// TwinCAT 3 PLC project Este_es_el_PLC
// ProgramVersion: 3.1.4024.0
// libraries:
//   Tc2_EtherCAT, * (Beckhoff Automation GmbH)
//   Tc2_ModbusSrv, * (Beckhoff Automation GmbH)
//   Tc2_Standard, * (Beckhoff Automation GmbH)
//   Tc2_System, * (Beckhoff Automation GmbH)
//   Tc2_Utilities, * (Beckhoff Automation GmbH)
//   Tc3_Module, * (Beckhoff Automation GmbH)
// project tree:
//   DUTs/ E_EventType.TcDUT, St_Event.TcDUT, ST_MachineStation.TcDUT (not stored)
//   GVLs/ GVL.TcGVL, Tags.TcGVL
//   / PlcTask.TcTTO
//   POUs/ conveyor1.TcPOU, MAIN.TcPOU
// real-time tasks:
//   TASK PlcTask: cycle T#10ms, priority 20, ADS port 350
//   TASK Device 1 (OPC UA Virtual)_Task_58: cycle T#40ms, priority 58, ADS port 351

CONFIGURATION Este_es_el_PLC
    RESOURCE PLC ON TwinCAT3
        TASK PlcTask(INTERVAL := T#10ms, PRIORITY := 20);
        PROGRAM MAIN WITH PlcTask : MAIN;
    END_RESOURCE
END_CONFIGURATION

// ---- DUTs/E_EventType.TcDUT
{attribute 'qualified_only'}
{attribute 'strict'}
TYPE E_EventType :
(
	alarm := 0,
	Message := 1
);
END_TYPE

// ---- DUTs/St_Event.TcDUT
TYPE St_Event :
STRUCT
	eEventType : E_EventType;
	eVentSeverity : TcEventSeverity;
	nEventIdentity : UDINT;
	SEventText : STRING(255);
	dtTimeStamp : DATE_AND_TIME;
END_STRUCT
END_TYPE

// ---- GVLs/GVL.TcGVL
{attribute 'qualified_only'}
VAR_GLOBAL
	mb_Input_Coils : ARRAY [0..255] OF BOOL;
	mb_Output_Coils : ARRAY [0..255] OF BOOL;
	mb_Input_Registers : ARRAY [0..255] OF WORD;
	mb_Output_Registers : ARRAY [0..255] OF WORD;
END_VAR

// ---- GVLs/Tags.TcGVL
{attribute 'qualified_only'}
VAR_GLOBAL
	bAutoMan : SR;
END_VAR

// ---- POUs/MAIN.TcPOU
PROGRAM MAIN
VAR
	bButtonStart,
	bButtonReset,
	bButtonStop: BOOL;
	bStatus : BOOL;
	bButtonLightStart,
	bButtonLightStop,
	bExtra, botroextra,bTercer,bCuarto : BOOL;
END_VAR

bButtonStart := GVL.mb_Output_Coils[0];
bButtonStop := GVL.mb_Output_Coils[1];
bButtonReset := GVL.mb_Output_Coils[29];
GVL.mb_Input_Coils[0] := bButtonLightStart;
GVL.mb_Input_Coils[1] := bButtonLightStop;
conveyor1();

Tags.bAutoMan(SET1 := bButtonStart, RESET := NOT bButtonStop);
bStatus := Tags.bAutoMan.Q1;
bButtonLightStart := bStatus;
bButtonLightStop := not bStatus;

END_PROGRAM

// ---- POUs/conveyor1.TcPOU
PROGRAM conveyor1
VAR
	bStatus: BOOL;
	bSensor2: BOOL;
	bSensor1: BOOL;
	bAlimentador1: BOOL;
	intCaseConveyor : INT;
	bButtonReset: BOOL;
	timer1, timer2, timer3,timer4 : TON;
	bConvFowar1: BOOL;
	bMachineCenterOpen: BOOL;
	bMachineCenterBusy: BOOL;
	bStartMachineCenter: BOOL;
	wMachineProgress: WORD;
END_VAR

bStatus := tags.bAutoMan.Q1;
bSensor1 := GVL.mb_Output_Coils[10];
bSensor2 := GVL.mb_Output_Coils[11];
bButtonReset := gvl.mb_Output_Coils[2];
bMachineCenterOpen := gvl.mb_Output_Coils[12];
bMachineCenterBusy := gvl.mb_Output_Coils[13];
wMachineProgress := gvl.mb_Output_Registers[0];


GVL.mb_Input_Coils[10] := bAlimentador1;
GVL.mb_Input_Coils[11] := bConvFowar1;
GVL.mb_Input_Coils[12] := bStartMachineCenter;

timer1(PT:= T#1S);
timer2(PT:= T#1S);
timer3(PT:= T#1S);


IF NOT bStatus THEN
	intCaseConveyor := 0;
END_IF

IF intCaseConveyor = 40 THEN
	timer2(IN := TRUE);
ELSE
	timer2(IN := FALSE);
END_IF

IF intCaseConveyor = 50 THEN
	timer3(IN := TRUE);
ELSE
	timer3(IN := FALSE);
END_IF

CASE intCaseConveyor OF
	00: timer1(IN:= FALSE);
		timer4(IN:= FALSE);
		bConvFowar1 := FALSE;
		bStartMachineCenter := False;
		IF bStatus THEN
			IF bSensor1 THEN
				intCaseConveyor := 10;
			ELSE
				intCaseConveyor := 20;
			END_IF
		END_IF
	10: IF bSensor1 THEN
			bAlimentador1 := TRUE;
		ELSE
			bAlimentador1 := FALSE;
			intCaseConveyor := 20;
		END_IF
	20: timer1(in:= TRUE);
		IF timer1.Q THEN
			bConvFowar1 := TRUE;
			intCaseConveyor := 30;
		END_IF;
	30: IF NOT bsensor2 THEN
			bConvFowar1 := FALSE;
				intCaseConveyor := 40;
		END_IF
		
	40: IF timer2.Q AND NOT bMachineCenterbusy  THEN
			bConvFowar1 := TRUE;
			IF bSensor2 THEN
				intCaseConveyor := 50;
			END_IF
		END_IF
	50: IF timer3.Q THEN
			bStartMachineCenter := TRUE;
			timer4(IN:= TRUE, PT:= T#300MS);
			IF timer4.Q THEN
				intCaseConveyor := 0;
			END_IF
		END_IF
		
END_CASE

END_PROGRAM
